// TIA Portal V17 export
// export: Created 2023-04-04T13:27:31.2861191Z, ExportSetting WithDefaults, DisplayName Totally Integrated Automation Portal, DisplayVersion V17, DisplayName TIA Portal Openness, DisplayVersion V17, DisplayName TIA Portal Version Control Interface, DisplayVersion V17, DisplayName STEP 7 Professional, DisplayVersion V17, DisplayName STEP 7 Safety, DisplayVersion V17, DisplayName WinCC Advanced, DisplayVersion V17
TYPE "typ_Config_Brightness_Sensor"
// stored: IsFailsafeCompliant false
   STRUCT
      ldt_ts : LDT;
      x_on : Bool;
      i_fps : Int;
   END_STRUCT;
END_TYPE
